// TIA Portal V18 export
FUNCTION_BLOCK "sirene_v2"   // FB7, FBD
{ S7_Optimized_Access := 'TRUE' }
VERSION : 0.1
// stored: AutoNumber true, IsIECCheckEnabled false, IsRetainMemResEnabled false, MemoryReserve 100, SetENOAutomatically false, UDAEnableTagReadback false
   VAR_INPUT
      bitStartUp : Bool;
   END_VAR
   VAR_OUTPUT
      sir_start : Bool;
      sirena_1 : Bool;
      sirena_2 : Bool;
      sirena_3 : Bool;
      sirena_4 : Bool;
      sirena_5 : Bool;
      sirena_6 : Bool;
   END_VAR
   VAR_IN_OUT
      greenTrigger : Bool;
      yellowTrigger : Bool;
      redTrigger : Bool;
      greenSettings : "UDT_settingsSirene";
      yellowSettings : "UDT_settingsSirene";
      redSettings : "UDT_settingsSirene";
   END_VAR
   VAR
      "step" : Int;
      fpBit_green : Bool;
      fpBit_yellow : Bool;
      fpBit_red : Bool;
      fpBit_greenTest : Bool;
      fpBit_yellowTest : Bool;
      fpBit_redTest : Bool;
      IEC_Timer_step1 { S7_SetPoint := 'True'} : IEC_TIMER;
      toneSelect : Int;
      toneDuration : Time;
      IEC_Timer_toneDuration { S7_SetPoint := 'True'} : IEC_TIMER;
      IEC_Timer_step2 { S7_SetPoint := 'True'} : IEC_TIMER;
      sirenaArray { ExternalAccessible := 'False'; ExternalVisible := 'False'; ExternalWritable := 'False'} : Array[0..15] of Bool;
   END_VAR
   VAR_TEMP   // added for the SCL form of the ladder/FBD networks
      _w1 : Bool;
      _w2 : Bool;
      _w3 : Bool;
      _w4 : Bool;
      _w5 : Bool;
      _w6 : Bool;
      _w7 : Bool;
      _w8 : Bool;
      _w9 : Bool;
      _w10 : Bool;
      _w11 : Bool;
      _w12 : Bool;
   END_VAR
BEGIN

REGION Network 2
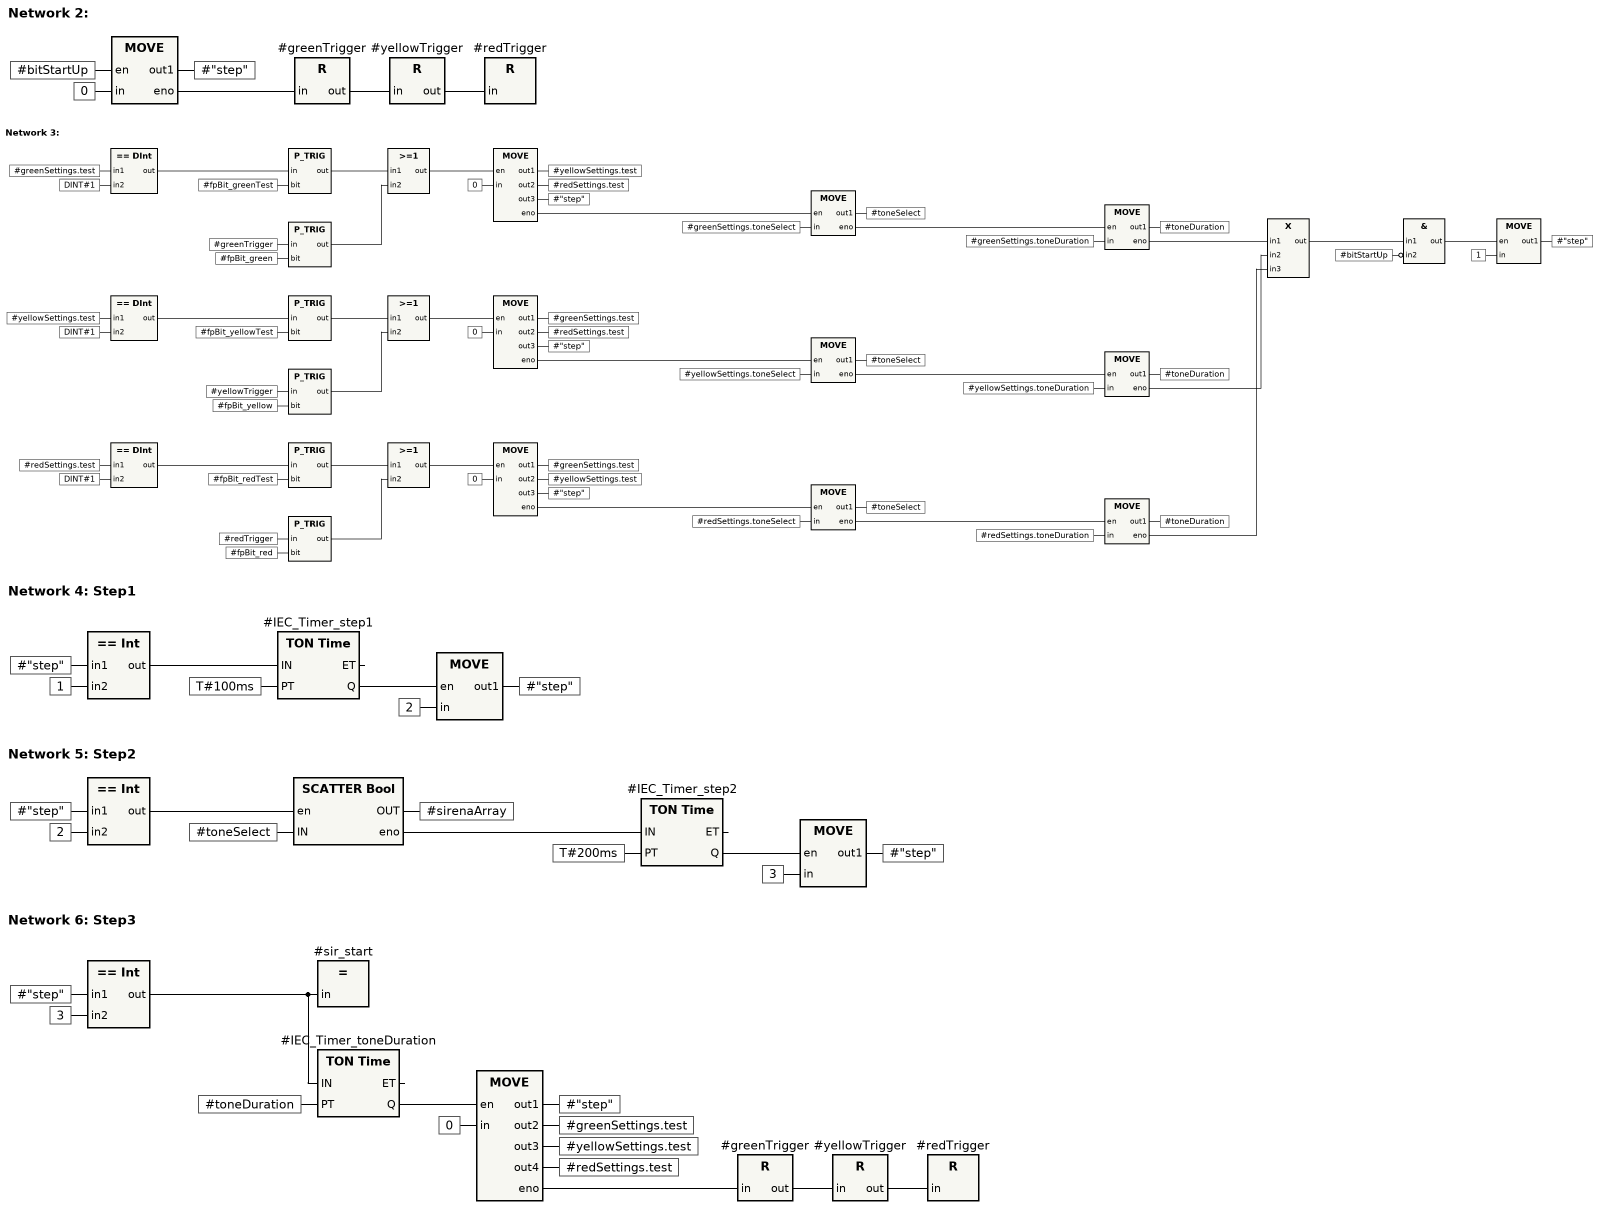
   IF #bitStartUp THEN
       #"step" := 0;
       #greenTrigger := FALSE;
       #yellowTrigger := FALSE;
       #redTrigger := FALSE;
   END_IF;
END_REGION

REGION Network 3
   #_w1 := #greenSettings.test = DINT#1;
   #_w2 := #_w1 AND NOT #fpBit_greenTest;   // rising edge
   #fpBit_greenTest := #_w1;
   #_w3 := #greenTrigger AND NOT #fpBit_green;   // rising edge
   #fpBit_green := #greenTrigger;
   #_w4 := #_w2 OR #_w3;
   IF #_w4 THEN
       #yellowSettings.test := 0;
       #redSettings.test := 0;
       #"step" := 0;
       #toneSelect := #greenSettings.toneSelect;
       #toneDuration := #greenSettings.toneDuration;
   END_IF;
   #_w5 := #yellowSettings.test = DINT#1;
   #_w6 := #_w5 AND NOT #fpBit_yellowTest;   // rising edge
   #fpBit_yellowTest := #_w5;
   #_w7 := #yellowTrigger AND NOT #fpBit_yellow;   // rising edge
   #fpBit_yellow := #yellowTrigger;
   #_w8 := #_w6 OR #_w7;
   IF #_w8 THEN
       #greenSettings.test := 0;
       #redSettings.test := 0;
       #"step" := 0;
       #toneSelect := #yellowSettings.toneSelect;
       #toneDuration := #yellowSettings.toneDuration;
   END_IF;
   #_w9 := #redSettings.test = DINT#1;
   #_w10 := #_w9 AND NOT #fpBit_redTest;   // rising edge
   #fpBit_redTest := #_w9;
   #_w11 := #redTrigger AND NOT #fpBit_red;   // rising edge
   #fpBit_red := #redTrigger;
   #_w12 := #_w10 OR #_w11;
   IF #_w12 THEN
       #greenSettings.test := 0;
       #yellowSettings.test := 0;
       #"step" := 0;
       #toneSelect := #redSettings.toneSelect;
       #toneDuration := #redSettings.toneDuration;
   END_IF;
   IF (#_w4 XOR #_w8 XOR #_w12) AND NOT #bitStartUp THEN #"step" := 1; END_IF;
END_REGION

REGION Network 4: Step1
   #IEC_Timer_step1.TON(IN := #"step" = 1, PT := T#100ms);
   IF #IEC_Timer_step1.Q THEN #"step" := 2; END_IF;
END_REGION

REGION Network 5: Step2
   #_w1 := #"step" = 2;
   SCATTER(EN := #_w1, IN := #toneSelect, OUT => #sirenaArray, ENO => #_w2);
   #IEC_Timer_step2.TON(IN := #_w2, PT := T#200ms);
   IF #IEC_Timer_step2.Q THEN #"step" := 3; END_IF;
END_REGION

REGION Network 6: Step3
   #sir_start := #"step" = 3;
   #IEC_Timer_toneDuration.TON(IN := #sir_start, PT := #toneDuration);
   IF #IEC_Timer_toneDuration.Q THEN
       #"step" := 0;
       #greenSettings.test := 0;
       #yellowSettings.test := 0;
       #redSettings.test := 0;
       #greenTrigger := FALSE;
       #yellowTrigger := FALSE;
       #redTrigger := FALSE;
   END_IF;
END_REGION

REGION Network 7: sirena_1
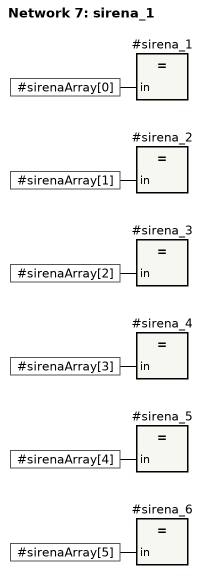
   #sirena_1 := #sirenaArray[0];
   #sirena_2 := #sirenaArray[1];
   #sirena_3 := #sirenaArray[2];
   #sirena_4 := #sirenaArray[3];
   #sirena_5 := #sirenaArray[4];
   #sirena_6 := #sirenaArray[5];
END_REGION
END_FUNCTION_BLOCK
